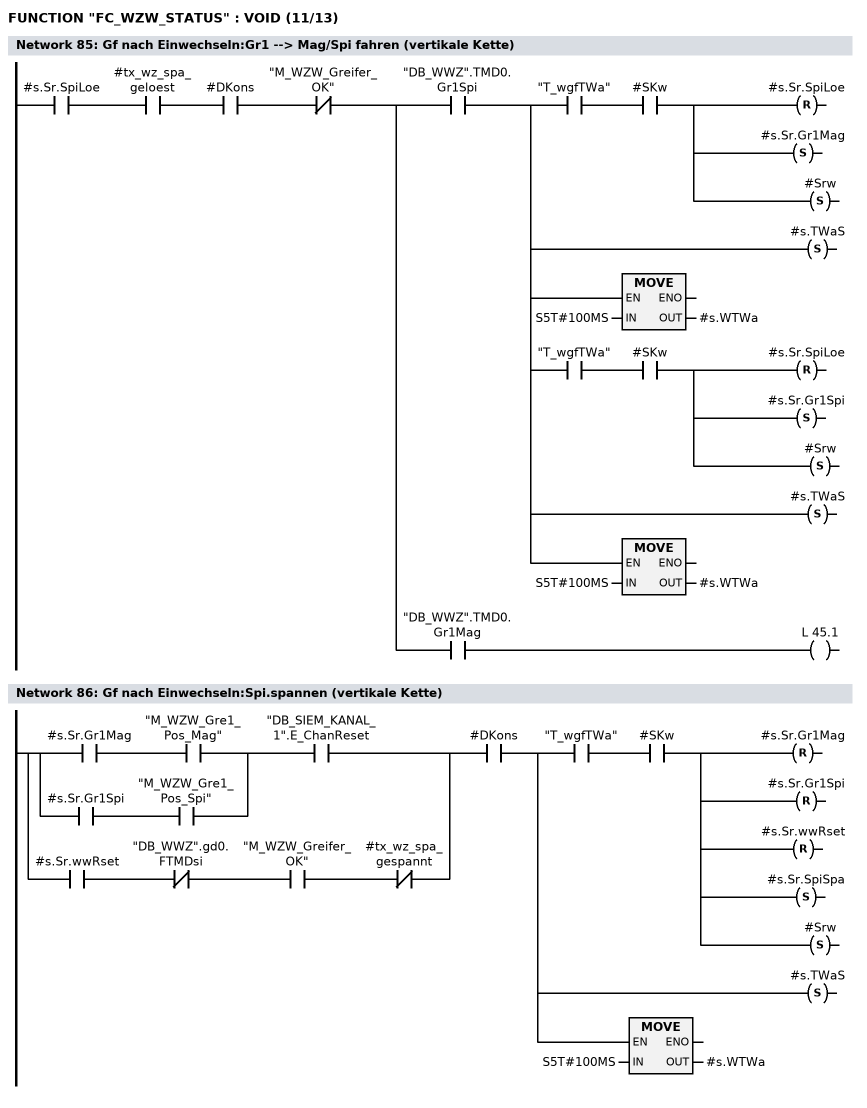

      U     #s.Sr.SpiLoe;
      U     #tx_wz_spa_geloest;
      U     #DKons;
      UN    "M_WZW_Greifer_OK";
      =     L     45.0;
      U     L     45.0;
      U     "DB_WWZ".TMD0.Gr1Spi;
      =     L     45.1;
      U     L     45.1;
      U     "T_wgfTWa";
      U     #SKw;
      R     #s.Sr.SpiLoe;
      S     #s.Sr.Gr1Mag;
      S     #Srw;
      U     L     45.1;
      BLD   102;
      S     #s.TWaS;
      U     L     45.1;
      SPBNB _023;
      L     S5T#100MS;
      T     #s.WTWa;
_023: NOP   0;
      U     L     45.0;
      U     "DB_WWZ".TMD0.Gr1Mag;
      =     L     45.1;
      U     L     45.1;
      U     "T_wgfTWa";
      U     #SKw;
      R     #s.Sr.SpiLoe;
      S     #s.Sr.Gr1Spi;
      S     #Srw;
      U     L     45.1;
      BLD   102;
      S     #s.TWaS;
      U     L     45.1;
      SPBNB _024;
      L     S5T#100MS;
      T     #s.WTWa;
_024: NOP   0;
NETWORK
TITLE =Gf nach Einwechseln:Spi.spannen (vertikale Kette)

      U(    ;
      U(    ;
      U     #s.Sr.Gr1Mag;
      U     "M_WZW_Gre1_Pos_Mag";
      O     ;
      U     #s.Sr.Gr1Spi;
      U     "M_WZW_Gre1_Pos_Spi";
      )     ;
      U     "DB_SIEM_KANAL_1".E_ChanReset;
      O     ;
      U     #s.Sr.wwRset;
      UN    "DB_WWZ".gd0.FTMDsi;
      U     "M_WZW_Greifer_OK";
      UN    #tx_wz_spa_gespannt;
      )     ;
      U     #DKons;
      =     L     45.0;
      U     L     45.0;
      U     "T_wgfTWa";
      U     #SKw;
      R     #s.Sr.Gr1Mag;
      R     #s.Sr.Gr1Spi;
      R     #s.Sr.wwRset;
      S     #s.Sr.SpiSpa;
      S     #Srw;
      U     L     45.0;
      BLD   102;
      S     #s.TWaS;
      U     L     45.0;
      SPBNB _025;
      L     S5T#100MS;
      T     #s.WTWa;
_025: NOP   0;
NETWORK
TITLE =Gf nach Einwechseln:umspeichern wenn schon Grf.ok & Spi.gespannt
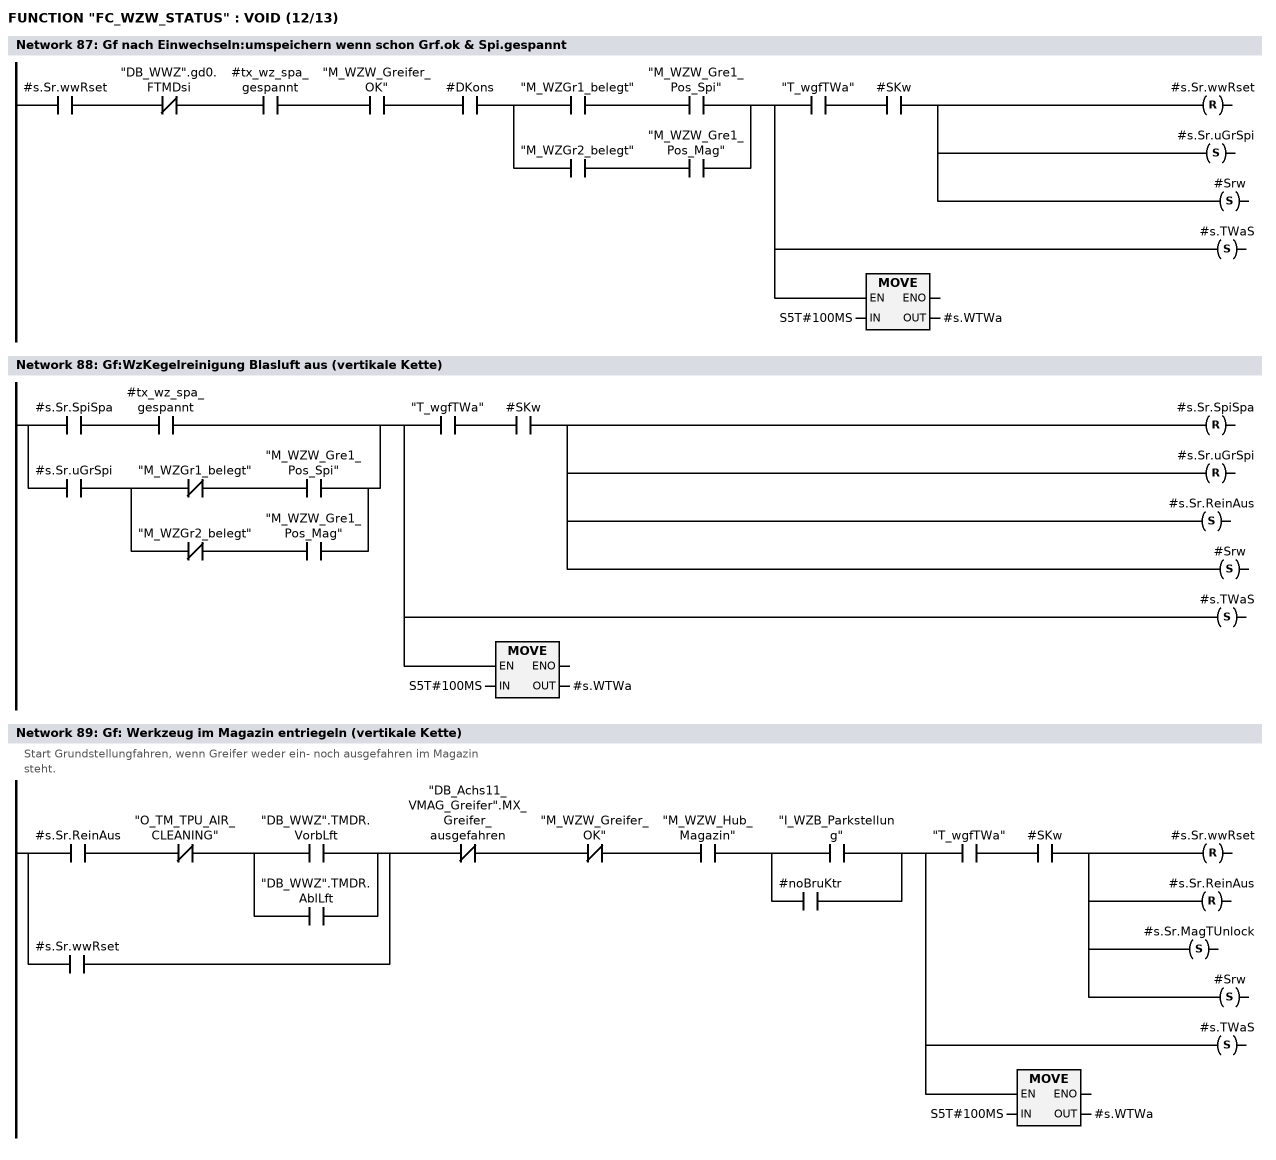

      U     #s.Sr.wwRset;
      UN    "DB_WWZ".gd0.FTMDsi;
      U     #tx_wz_spa_gespannt;
      U     "M_WZW_Greifer_OK";
      U     #DKons;
      U(    ;
      U     "M_WZGr1_belegt";
      U     "M_WZW_Gre1_Pos_Spi";
      O     ;
      U     "M_WZGr2_belegt";
      U     "M_WZW_Gre1_Pos_Mag";
      )     ;
      =     L     45.0;
      U     L     45.0;
      U     "T_wgfTWa";
      U     #SKw;
      R     #s.Sr.wwRset;
      S     #s.Sr.uGrSpi;
      S     #Srw;
      U     L     45.0;
      BLD   102;
      S     #s.TWaS;
      U     L     45.0;
      SPBNB _026;
      L     S5T#100MS;
      T     #s.WTWa;
_026: NOP   0;
NETWORK
TITLE =Gf:WzKegelreinigung Blasluft aus (vertikale Kette)

      U     #s.Sr.SpiSpa;
      U     #tx_wz_spa_gespannt;
      O     ;
      U     #s.Sr.uGrSpi;
      U(    ;
      UN    "M_WZGr1_belegt";
      U     "M_WZW_Gre1_Pos_Spi";
      O     ;
      UN    "M_WZGr2_belegt";
      U     "M_WZW_Gre1_Pos_Mag";
      )     ;
      =     L     45.0;
      U     L     45.0;
      U     "T_wgfTWa";
      U     #SKw;
      R     #s.Sr.SpiSpa;
      R     #s.Sr.uGrSpi;
      S     #s.Sr.ReinAus;
      S     #Srw;
      U     L     45.0;
      BLD   102;
      S     #s.TWaS;
      U     L     45.0;
      SPBNB _027;
      L     S5T#100MS;
      T     #s.WTWa;
_027: NOP   0;
NETWORK
TITLE =Gf: Werkzeug im Magazin entriegeln (vertikale Kette)
//Start Grundstellungfahren, wenn Greifer weder ein- noch ausgefahren im Magazin
//steht.
      U(    ;
      U     #s.Sr.ReinAus;
      UN    "O_TM_TPU_AIR_CLEANING";
      U(    ;
      O     "DB_WWZ".TMDR.VorbLft;
      O     "DB_WWZ".TMDR.AblLft;
      )     ;
      O     #s.Sr.wwRset;
      )     ;
      UN    "DB_Achs11_VMAG_Greifer".MX_Greifer_ausgefahren;
      UN    "M_WZW_Greifer_OK";
      U     "M_WZW_Hub_Magazin";
      U(    ;
      O     "I_WZB_Parkstellung";
      O     #noBruKtr;
      )     ;
      =     L     45.0;
      U     L     45.0;
      U     "T_wgfTWa";
      U     #SKw;
      R     #s.Sr.wwRset;
      R     #s.Sr.ReinAus;
      S     #s.Sr.MagTUnlock;
      S     #Srw;
      U     L     45.0;
      BLD   102;
      S     #s.TWaS;
      U     L     45.0;
      SPBNB _028;
      L     S5T#100MS;
      T     #s.WTWa;
_028: NOP   0;
NETWORK
TITLE =Gf: Greifer ausfahren (vertikale Kette)
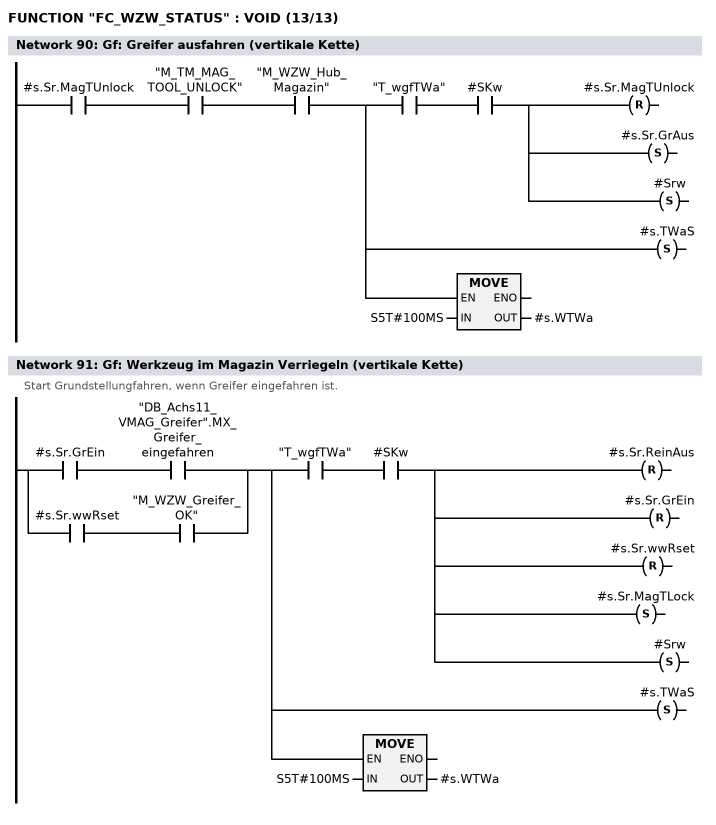

      U     #s.Sr.MagTUnlock;
      U     "M_TM_MAG_TOOL_UNLOCK";
      U     "M_WZW_Hub_Magazin";
      =     L     45.0;
      U     L     45.0;
      U     "T_wgfTWa";
      U     #SKw;
      R     #s.Sr.MagTUnlock;
      S     #s.Sr.GrAus;
      S     #Srw;
      U     L     45.0;
      BLD   102;
      S     #s.TWaS;
      U     L     45.0;
      SPBNB _029;
      L     S5T#100MS;
      T     #s.WTWa;
_029: NOP   0;
NETWORK
TITLE =Gf: Werkzeug im Magazin Verriegeln (vertikale Kette)
//Start Grundstellungfahren, wenn Greifer eingefahren ist.
      U     #s.Sr.GrEin;
      U     "DB_Achs11_VMAG_Greifer".MX_Greifer_eingefahren;
      O     ;
      U     #s.Sr.wwRset;
      U     "M_WZW_Greifer_OK";
      =     L     45.0;
      U     L     45.0;
      U     "T_wgfTWa";
      U     #SKw;
      R     #s.Sr.ReinAus;
      R     #s.Sr.GrEin;
      R     #s.Sr.wwRset;
      S     #s.Sr.MagTLock;
      S     #Srw;
      U     L     45.0;
      BLD   102;
      S     #s.TWaS;
      U     L     45.0;
      SPBNB _02a;
      L     S5T#100MS;
      T     #s.WTWa;
_02a: NOP   0;
NETWORK
TITLE =Gf: Querhub in Grundstellung fahren (vertikale Kette)

      U     #s.Sr.MagTLock;
      U     "M_TM_MAG_TOOL_LOCK";
      U     "M_WZW_Greifer_OK";
      O     ;
      U     #s.Sr.GrAus;
      U     "DB_Achs11_VMAG_Greifer".MX_Greifer_ausgefahren;
      =     L     44.0;
      U     L     44.0;
      U     "T_wgfTWa";
      U     #SKw;
      =     L     44.1;
      O     L     44.1;
      O     "DB_OEM".WZW_in_Grdst;
      R     #s.Sr.MagTLock;
      R     #s.Sr.GrAus;
      U     L     44.1;
      BLD   102;
      S     #Srw;
      U     L     44.1;
      BLD   102;
      S     #s.Sr.WzHubGf;
      U     L     44.0;
      BLD   102;
      S     #s.TWaS;
      U     L     44.0;
      SPBNB _051;
      L     S5T#100MS;
      T     #s.WTWa;
_051: NOP   0;
NETWORK
TITLE =Gf: Greifer einfahren (vertikale Kette)
//Start Grundstellungfahren, wenn der Greifer weder ein- noch ausgefahren und der
//querhub in Grundstellung ist.
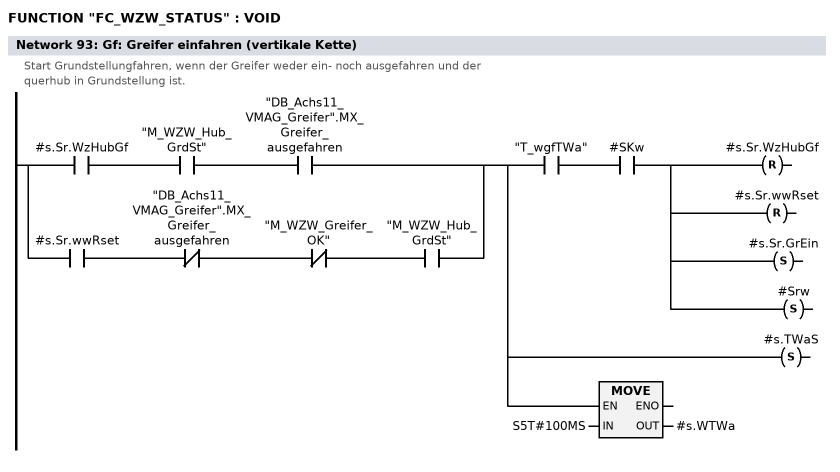
      U     #s.Sr.WzHubGf;
      U     "M_WZW_Hub_GrdSt";
      U     "DB_Achs11_VMAG_Greifer".MX_Greifer_ausgefahren;
      O     ;
      U     #s.Sr.wwRset;
      UN    "DB_Achs11_VMAG_Greifer".MX_Greifer_ausgefahren;
      UN    "M_WZW_Greifer_OK";
      U     "M_WZW_Hub_GrdSt";
      =     L     45.0;
      U     L     45.0;
      U     "T_wgfTWa";
      U     #SKw;
      R     #s.Sr.WzHubGf;
      R     #s.Sr.wwRset;
      S     #s.Sr.GrEin;
      S     #Srw;
      U     L     45.0;
      BLD   102;
      S     #s.TWaS;
      U     L     45.0;
      SPBNB _02b;
      L     S5T#100MS;
      T     #s.WTWa;
_02b: NOP   0;
NETWORK
TITLE =----- Ende vertikale Kette -----

E_VK: NOP   0;

NETWORK
TITLE =Gf: X-Achse zum Arbeitsraum

      U     #s.Sr.WzwvGf;
      U(    ;
      O     "I_WW_Rueck_hlt_GST";
      O     "M_WZM_Regal_angewaehlt";
      )     ;
      O     ;
      U     #s.Sr.WzHubGf;
      U     "M_WZW_Hub_GrdSt";
      O     ;
      U     #s.Sr.GrEin;
      U     "DB_Achs11_VMAG_Greifer".MX_Greifer_eingefahren;
      O     ;
      U     #s.Sr.ReinAus;
      UN    "O_TM_TPU_AIR_CLEANING";
      =     L     44.0;
      U     L     44.0;
      U     "T_wgfTWa";
      U     #SKw;
      =     L     44.1;
      O     L     44.1;
      O     "DB_OEM".WZW_in_Grdst;
      R     #s.Sr.WzwvGf;
      R     #s.Sr.WzHubGf;
      R     #s.Sr.GrEin;
      R     #s.Sr.ReinAus;
      U     L     44.1;
      BLD   102;
      S     #s.Sr.XArbRaum;
      U     L     44.1;
      BLD   102;
      S     #Srw;
      U     L     44.0;
      BLD   102;
      S     #s.TWaS;
      U     L     44.0;
      SPBNB _053;
      L     S5T#100MS;
      T     #s.WTWa;
_053: NOP   0;
NETWORK
TITLE =Gf: Wzw-Tür schliessen
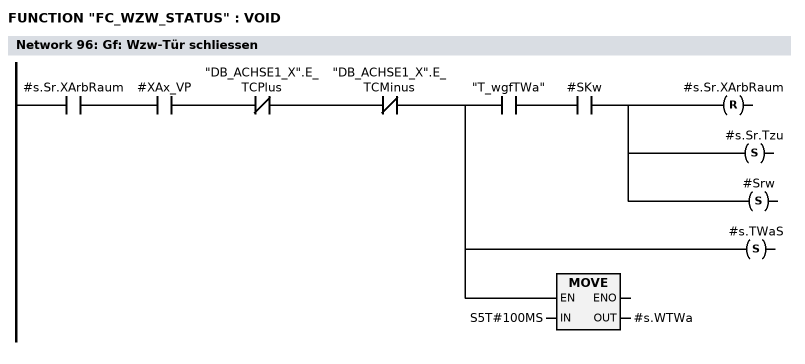

      U     #s.Sr.XArbRaum;
      U     #XAx_VP;
      UN    "DB_ACHSE1_X".E_TCPlus;
      UN    "DB_ACHSE1_X".E_TCMinus;
      =     L     45.0;
      U     L     45.0;
      U     "T_wgfTWa";
      U     #SKw;
      R     #s.Sr.XArbRaum;
      S     #s.Sr.Tzu;
      S     #Srw;
      U     L     45.0;
      BLD   102;
      S     #s.TWaS;
      U     L     45.0;
      SPBNB _02c;
      L     S5T#100MS;
      T     #s.WTWa;
_02c: NOP   0;
NETWORK
TITLE =Gf fertig, Ende SrKette
//Schritt muss auch ohne Weiterschaltbedingung beendet werden, da sonst im
//Einzelschritt der Schritt gesetzt bleibt.
//Grund: Wenn Werkzeugwechsler in Grundstellung ist wird kein Startimpuls
//mehr ausgeloest.
      U     #s.Sr.Tzu;
      U     "I_WW_1_Klappe_zu";
      UN    "I_WW_1_Klappe_auf";
      =     L     44.0;
      U     L     44.0;
      U     "T_wgfTWa";
      U     #SKw;
      =     L     44.1;
      O     L     44.1;
      O     "DB_OEM".WZW_in_Grdst;
      R     #s.Sr.Tzu;
      R     #s.Sr.GrEin;
      R     #s.Sr.WzHubGf;
      U     L     44.1;
      BLD   102;
      S     #Srw;
      U     L     44.0;
      BLD   102;
      S     #s.TWaS;
      U     L     44.0;
      SPBNB _055;
      L     S5T#100MS;
      T     #s.WTWa;
_055: NOP   0;
NETWORK
TITLE =Ansteuerung Wartezeit TWa
//Verweilzeit zwischen den Schritten der Schrittkette
//Die Zeitbasis wird jeweils über #WTWa übergeben!
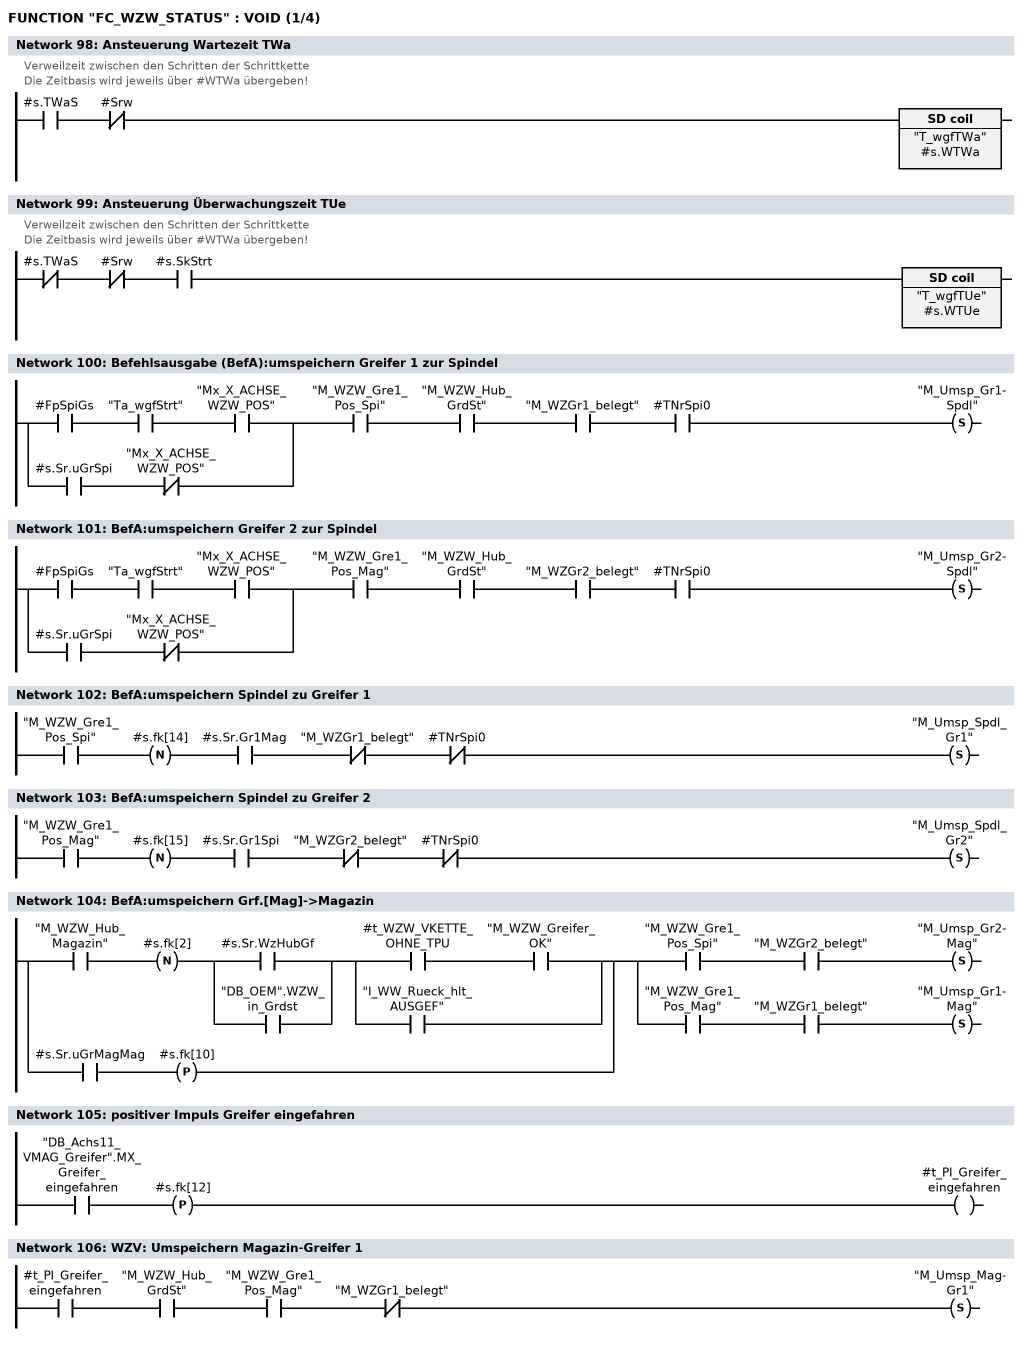
      U     #s.TWaS;
      UN    #Srw;
      L     #s.WTWa;
      SE    "T_wgfTWa";
NETWORK
TITLE =Ansteuerung Überwachungszeit TUe
//Verweilzeit zwischen den Schritten der Schrittkette
//Die Zeitbasis wird jeweils über #WTWa übergeben!
      UN    #s.TWaS;
      UN    #Srw;
      U     #s.SkStrt;
      L     #s.WTUe;
      SE    "T_wgfTUe";
NETWORK
TITLE =Befehlsausgabe (BefA):umspeichern Greifer 1 zur Spindel

      U(    ;
      U     #FpSpiGs;
      U     "Ta_wgfStrt";
      U     "Mx_X_ACHSE_WZW_POS";
      O     ;
      U     #s.Sr.uGrSpi;
      UN    "Mx_X_ACHSE_WZW_POS";
      )     ;
      U     "M_WZW_Gre1_Pos_Spi";
      U     "M_WZW_Hub_GrdSt";
      U     "M_WZGr1_belegt";
      U     #TNrSpi0;
      S     "M_Umsp_Gr1-Spdl";
NETWORK
TITLE =BefA:umspeichern Greifer 2 zur Spindel

      U(    ;
      U     #FpSpiGs;
      U     "Ta_wgfStrt";
      U     "Mx_X_ACHSE_WZW_POS";
      O     ;
      U     #s.Sr.uGrSpi;
      UN    "Mx_X_ACHSE_WZW_POS";
      )     ;
      U     "M_WZW_Gre1_Pos_Mag";
      U     "M_WZW_Hub_GrdSt";
      U     "M_WZGr2_belegt";
      U     #TNrSpi0;
      S     "M_Umsp_Gr2-Spdl";
NETWORK
TITLE =BefA:umspeichern Spindel zu Greifer 1

      U     "M_WZW_Gre1_Pos_Spi";
      FN    #s.fk[14];
      U     #s.Sr.Gr1Mag;
      UN    "M_WZGr1_belegt";
      UN    #TNrSpi0;
      S     "M_Umsp_Spdl_Gr1";
NETWORK
TITLE =BefA:umspeichern Spindel zu Greifer 2

      U     "M_WZW_Gre1_Pos_Mag";
      FN    #s.fk[15];
      U     #s.Sr.Gr1Spi;
      UN    "M_WZGr2_belegt";
      UN    #TNrSpi0;
      S     "M_Umsp_Spdl_Gr2";
NETWORK
TITLE =BefA:umspeichern Grf.[Mag]->Magazin

      U     "M_WZW_Hub_Magazin";
      FN    #s.fk[2];
      U(    ;
      O     #s.Sr.WzHubGf;
      O     "DB_OEM".WZW_in_Grdst;
      )     ;
      U(    ;
      U     #t_WZW_VKETTE_OHNE_TPU;
      U     "M_WZW_Greifer_OK";
      O     "I_WW_Rueck_hlt_AUSGEF";
      )     ;
      O(    ;
      U     #s.Sr.uGrMagMag;
      FP    #s.fk[10];
      )     ;
      =     L     45.0;
      U     L     45.0;
      U     "M_WZW_Gre1_Pos_Spi";
      U     "M_WZGr2_belegt";
      S     "M_Umsp_Gr2-Mag";
      U     L     45.0;
      U     "M_WZW_Gre1_Pos_Mag";
      U     "M_WZGr1_belegt";
      S     "M_Umsp_Gr1-Mag";
NETWORK
TITLE =positiver Impuls Greifer eingefahren

      U     "DB_Achs11_VMAG_Greifer".MX_Greifer_eingefahren;
      FP    #s.fk[12];
      =     #t_PI_Greifer_eingefahren;
NETWORK
TITLE =WZV: Umspeichern Magazin-Greifer 1

      U     #t_PI_Greifer_eingefahren;
      U     "M_WZW_Hub_GrdSt";
      U     "M_WZW_Gre1_Pos_Mag";
      UN    "M_WZGr1_belegt";
      S     "M_Umsp_Mag-Gr1";
NETWORK
TITLE =WZV: Umspeichern Magazin-Greifer 2
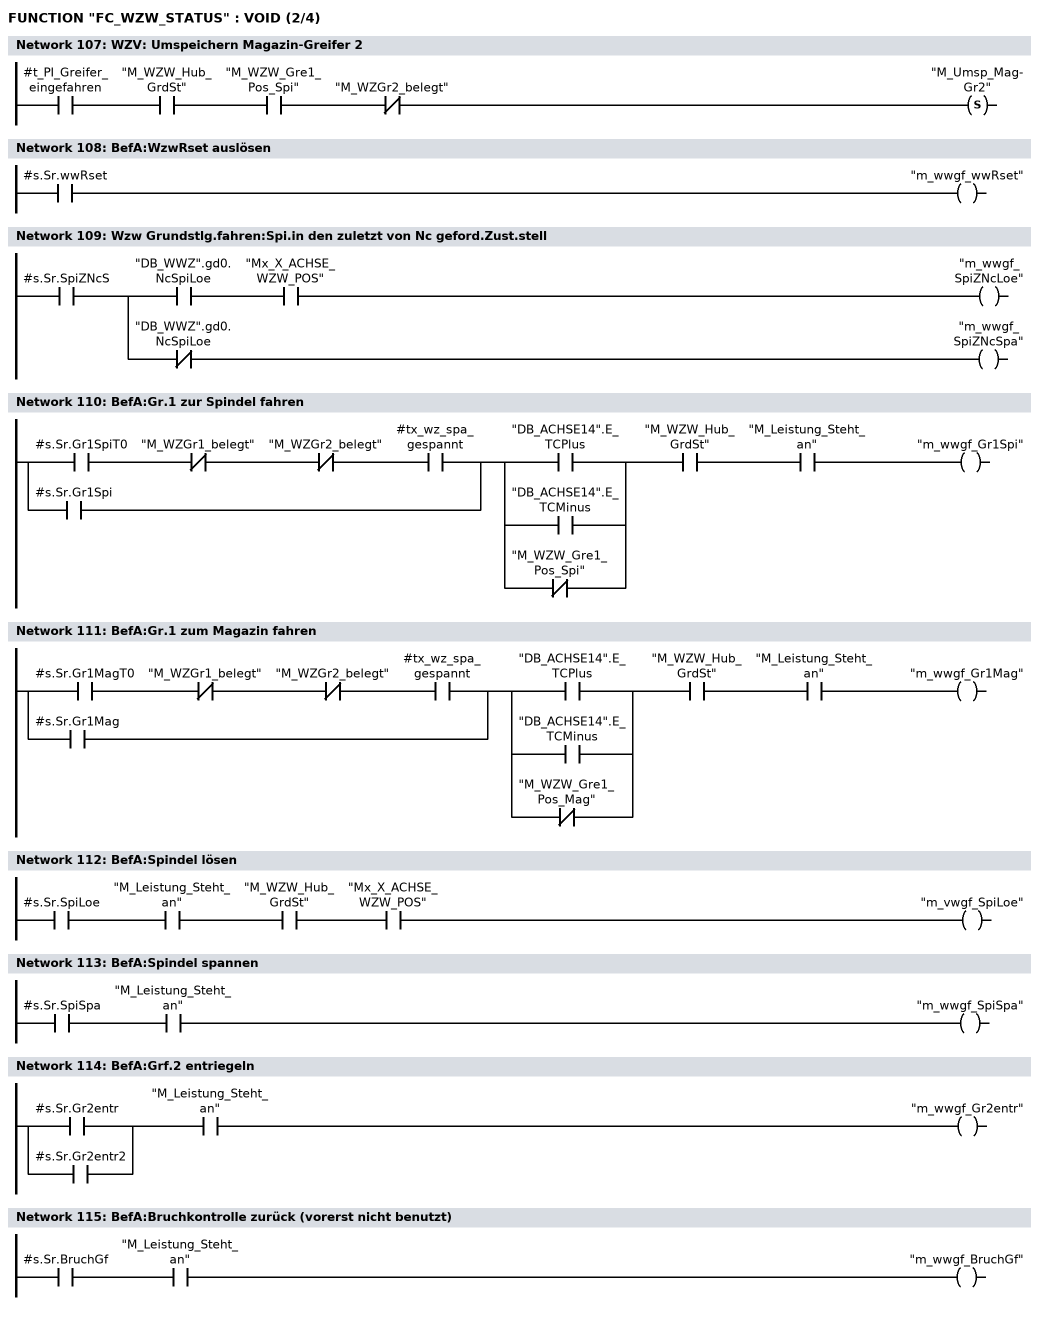

      U     #t_PI_Greifer_eingefahren;
      U     "M_WZW_Hub_GrdSt";
      U     "M_WZW_Gre1_Pos_Spi";
      UN    "M_WZGr2_belegt";
      S     "M_Umsp_Mag-Gr2";
NETWORK
TITLE =BefA:WzwRset auslösen

      U     #s.Sr.wwRset;
      =     "m_wwgf_wwRset";
NETWORK
TITLE =Wzw Grundstlg.fahren:Spi.in den zuletzt von Nc geford.Zust.stell

      U     #s.Sr.SpiZNcS;
      =     L     45.0;
      U     L     45.0;
      U     "DB_WWZ".gd0.NcSpiLoe;
      U     "Mx_X_ACHSE_WZW_POS";
      =     "m_wwgf_SpiZNcLoe";
      U     L     45.0;
      UN    "DB_WWZ".gd0.NcSpiLoe;
      =     "m_wwgf_SpiZNcSpa";
NETWORK
TITLE =BefA:Gr.1 zur Spindel fahren

      U(    ;
      U     #s.Sr.Gr1SpiT0;
      UN    "M_WZGr1_belegt";
      UN    "M_WZGr2_belegt";
      U     #tx_wz_spa_gespannt;
      O     #s.Sr.Gr1Spi;
      )     ;
      U(    ;
      O     "DB_ACHSE14".E_TCPlus;
      O     "DB_ACHSE14".E_TCMinus;
      ON    "M_WZW_Gre1_Pos_Spi";
      )     ;
      U     "M_WZW_Hub_GrdSt";
      U     "M_Leistung_Steht_an";
      =     "m_wwgf_Gr1Spi";
NETWORK
TITLE =BefA:Gr.1 zum Magazin fahren

      U(    ;
      U     #s.Sr.Gr1MagT0;
      UN    "M_WZGr1_belegt";
      UN    "M_WZGr2_belegt";
      U     #tx_wz_spa_gespannt;
      O     #s.Sr.Gr1Mag;
      )     ;
      U(    ;
      O     "DB_ACHSE14".E_TCPlus;
      O     "DB_ACHSE14".E_TCMinus;
      ON    "M_WZW_Gre1_Pos_Mag";
      )     ;
      U     "M_WZW_Hub_GrdSt";
      U     "M_Leistung_Steht_an";
      =     "m_wwgf_Gr1Mag";
NETWORK
TITLE =BefA:Spindel lösen

      U     #s.Sr.SpiLoe;
      U     "M_Leistung_Steht_an";
      U     "M_WZW_Hub_GrdSt";
      U     "Mx_X_ACHSE_WZW_POS";
      =     "m_vwgf_SpiLoe";
NETWORK
TITLE =BefA:Spindel spannen

      U     #s.Sr.SpiSpa;
      U     "M_Leistung_Steht_an";
      =     "m_wwgf_SpiSpa";
NETWORK
TITLE =BefA:Grf.2 entriegeln

      U(    ;
      O     #s.Sr.Gr2entr;
      O     #s.Sr.Gr2entr2;
      )     ;
      U     "M_Leistung_Steht_an";
      =     "m_wwgf_Gr2entr";
NETWORK
TITLE =BefA:Bruchkontrolle zurück (vorerst nicht benutzt)

      U     #s.Sr.BruchGf;
      U     "M_Leistung_Steht_an";
      =     "m_wwgf_BruchGf";
NETWORK
TITLE =BefA:Wz-Reinigung zurück
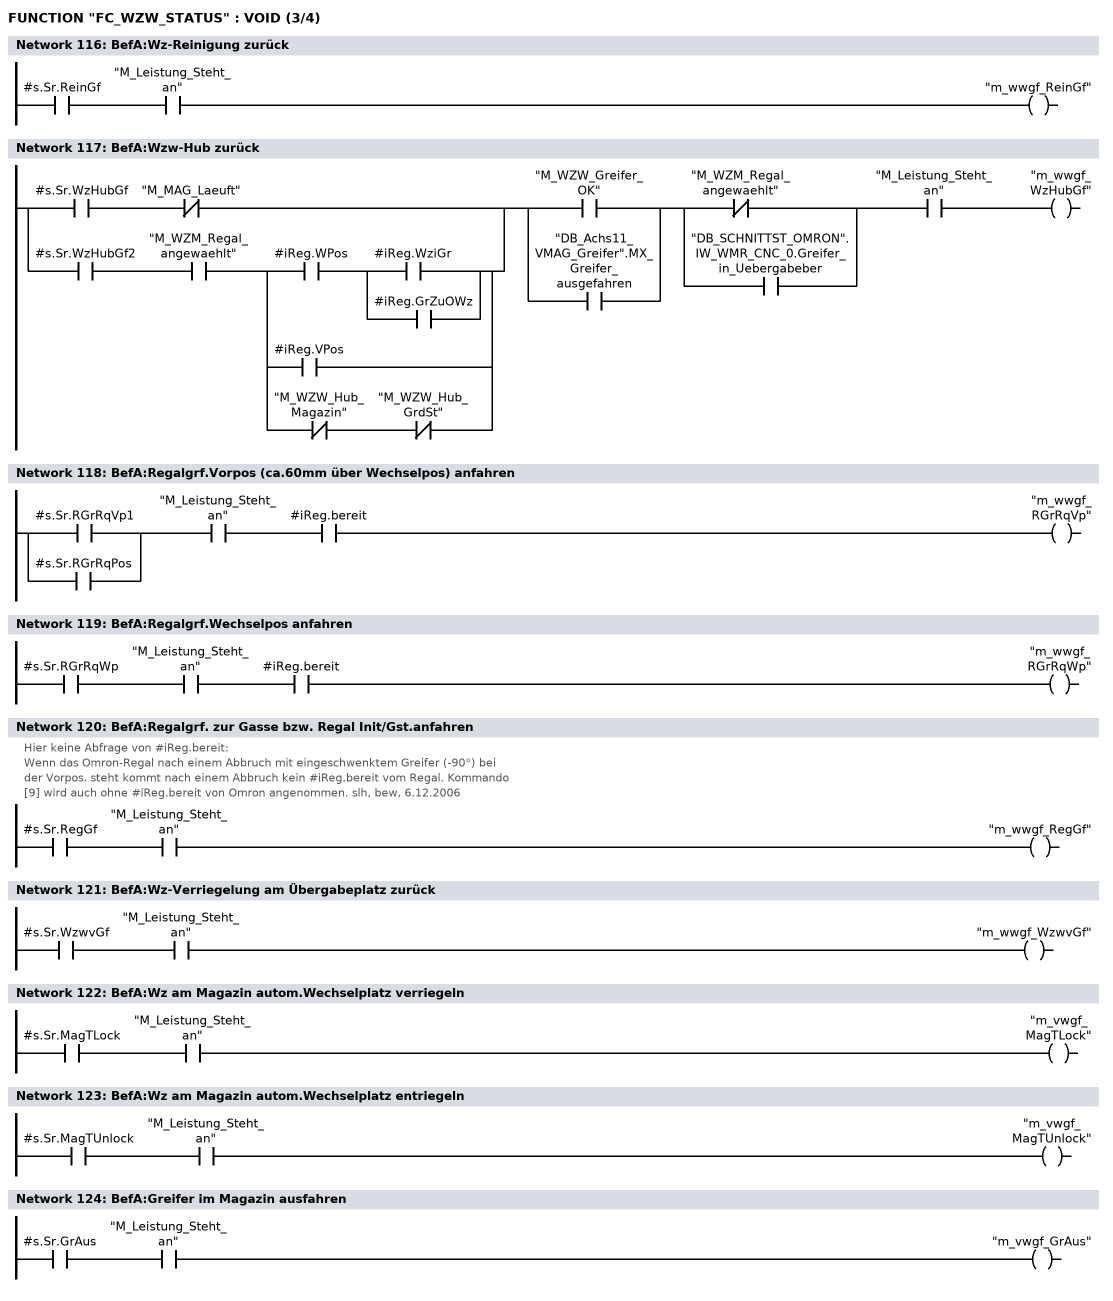

      U     #s.Sr.ReinGf;
      U     "M_Leistung_Steht_an";
      =     "m_wwgf_ReinGf";
NETWORK
TITLE =BefA:Wzw-Hub zurück

      U(    ;
      U     #s.Sr.WzHubGf;
      UN    "M_MAG_Laeuft";
      O     ;
      U     #s.Sr.WzHubGf2;
      U     "M_WZM_Regal_angewaehlt";
      U(    ;
      U     #iReg.WPos;
      U(    ;
      O     #iReg.WziGr;
      O     #iReg.GrZuOWz;
      )     ;
      O     #iReg.VPos;
      O     ;
      UN    "M_WZW_Hub_Magazin";
      UN    "M_WZW_Hub_GrdSt";
      )     ;
      )     ;
      U(    ;
      O     "M_WZW_Greifer_OK";
      O     "DB_Achs11_VMAG_Greifer".MX_Greifer_ausgefahren;
      )     ;
      U(    ;
      ON    "M_WZM_Regal_angewaehlt";
      O     "DB_SCHNITTST_OMRON".IW_WMR_CNC_0.Greifer_in_Uebergabeber;
      )     ;
      U     "M_Leistung_Steht_an";
      =     "m_wwgf_WzHubGf";
NETWORK
TITLE =BefA:Regalgrf.Vorpos (ca.60mm über Wechselpos) anfahren

      U(    ;
      O     #s.Sr.RGrRqVp1;
      O     #s.Sr.RGrRqPos;
      )     ;
      U     "M_Leistung_Steht_an";
      U     #iReg.bereit;
      =     "m_wwgf_RGrRqVp";
NETWORK
TITLE =BefA:Regalgrf.Wechselpos anfahren

      U     #s.Sr.RGrRqWp;
      U     "M_Leistung_Steht_an";
      U     #iReg.bereit;
      =     "m_wwgf_RGrRqWp";
NETWORK
TITLE =BefA:Regalgrf. zur Gasse bzw. Regal Init/Gst.anfahren
//Hier keine Abfrage von #iReg.bereit:
//Wenn das Omron-Regal nach einem Abbruch mit eingeschwenktem Greifer (-90°) bei
//der Vorpos. steht kommt nach einem Abbruch kein #iReg.bereit vom Regal. Kommando
//[9] wird auch ohne #iReg.bereit von Omron angenommen. slh, bew, 6.12.2006
      U     #s.Sr.RegGf;
      U     "M_Leistung_Steht_an";
      =     "m_wwgf_RegGf";
NETWORK
TITLE =BefA:Wz-Verriegelung am Übergabeplatz zurück

      U     #s.Sr.WzwvGf;
      U     "M_Leistung_Steht_an";
      =     "m_wwgf_WzwvGf";
NETWORK
TITLE =BefA:Wz am Magazin autom.Wechselplatz verriegeln

      U     #s.Sr.MagTLock;
      U     "M_Leistung_Steht_an";
      =     "m_vwgf_MagTLock";
NETWORK
TITLE =BefA:Wz am Magazin autom.Wechselplatz entriegeln

      U     #s.Sr.MagTUnlock;
      U     "M_Leistung_Steht_an";
      =     "m_vwgf_MagTUnlock";
NETWORK
TITLE =BefA:Greifer im Magazin ausfahren

      U     #s.Sr.GrAus;
      U     "M_Leistung_Steht_an";
      =     "m_vwgf_GrAus";
NETWORK
TITLE =BefA:Greifer im Magazin einfahren
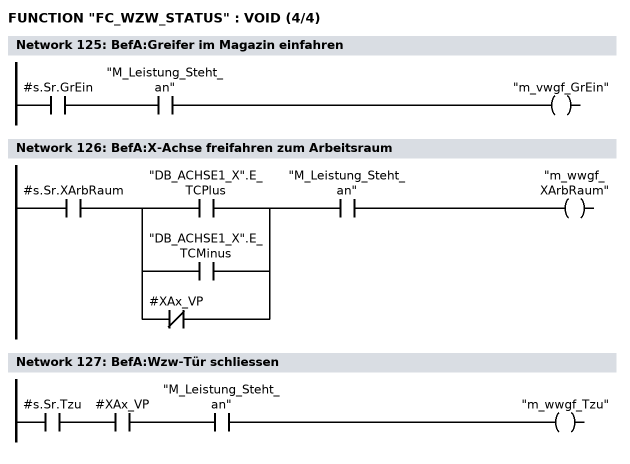

      U     #s.Sr.GrEin;
      U     "M_Leistung_Steht_an";
      =     "m_vwgf_GrEin";
NETWORK
TITLE =BefA:X-Achse freifahren zum Arbeitsraum

      U     #s.Sr.XArbRaum;
      U(    ;
      O     "DB_ACHSE1_X".E_TCPlus;
      O     "DB_ACHSE1_X".E_TCMinus;
      ON    #XAx_VP;
      )     ;
      U     "M_Leistung_Steht_an";
      =     "m_wwgf_XArbRaum";
NETWORK
TITLE =BefA:Wzw-Tür schliessen

      U     #s.Sr.Tzu;
      U     #XAx_VP;
      U     "M_Leistung_Steht_an";
      =     "m_wwgf_Tzu";
NETWORK
TITLE =BefA:Halt Asup

      UN    "DB_ASUP_MACHINE".Start_Asup;
      R     "m_vwgf_stpAsup1";
      UN    "m_wwgf_XArbRaum";
      UN    "m_wwgf_Gr1Spi";
      UN    "m_wwgf_Gr1Mag";
      UN(   ;
      U     "IX_MSST_Ta_2_4";
      UN    "M_Handbetrieb";
      )     ;
      FP    #s.fk[7];
      S     "m_vwgf_stpAsup1";
      NOP   0;
NETWORK
TITLE =Bedienungshinweise
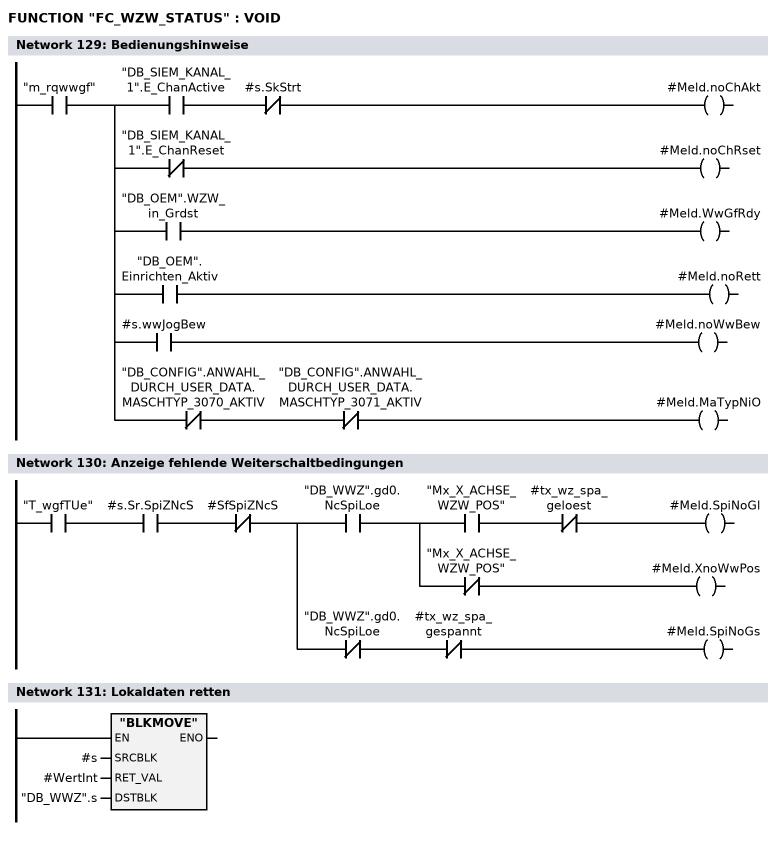

      U     "m_rqwwgf";
      =     L     45.0;
      U     L     45.0;
      U     "DB_SIEM_KANAL_1".E_ChanActive;
      UN    #s.SkStrt;
      =     #Meld.noChAkt;
      U     L     45.0;
      UN    "DB_SIEM_KANAL_1".E_ChanReset;
      =     #Meld.noChRset;
      U     L     45.0;
      U     "DB_OEM".WZW_in_Grdst;
      =     #Meld.WwGfRdy;
      U     L     45.0;
      U     "DB_OEM".Einrichten_Aktiv;
      =     #Meld.noRett;
      U     L     45.0;
      U     #s.wwJogBew;
      =     #Meld.noWwBew;
      U     L     45.0;
      UN    "DB_CONFIG".ANWAHL_DURCH_USER_DATA.MASCHTYP_3070_AKTIV;
      UN    "DB_CONFIG".ANWAHL_DURCH_USER_DATA.MASCHTYP_3071_AKTIV;
      =     #Meld.MaTypNiO;
NETWORK
TITLE =Anzeige fehlende Weiterschaltbedingungen

      U     "T_wgfTUe";
      U     #s.Sr.SpiZNcS;
      UN    #SfSpiZNcS;
      =     L     45.0;
      U     L     45.0;
      U     "DB_WWZ".gd0.NcSpiLoe;
      =     L     45.1;
      U     L     45.1;
      U     "Mx_X_ACHSE_WZW_POS";
      UN    #tx_wz_spa_geloest;
      =     #Meld.SpiNoGl;
      U     L     45.1;
      UN    "Mx_X_ACHSE_WZW_POS";
      =     #Meld.XnoWwPos;
      U     L     45.0;
      UN    "DB_WWZ".gd0.NcSpiLoe;
      UN    #tx_wz_spa_gespannt;
      =     #Meld.SpiNoGs;
NETWORK
TITLE =Lokaldaten retten

      CALL "BLKMOVE" (
           SRCBLK                   := #s,
           RET_VAL                  := #WertInt,
           DSTBLK                   := "DB_WWZ".s);
      NOP   0;
END_FUNCTION

